// TIA Portal project "Data Logging Test 2_V17" (V17)

(* hardware
DEVICE "S7-1200 station_1"  S7-1200 Station
   slot 0: "Rack_0"  S7-1200 Rack  Rack  V1.0
   slot 1: "PLC_Wind Project-Datalogging"  CPU 1214C DC/DC/DC  6ES7 214-1AG40-0XB0  V4.2
   slot 2: "AI 4x13BIT/AQ 2x14BIT_1"  6ES7 234-4HE32-0XB0  V2.1
*)

// ===== PLC "PLC_Wind Project-Datalogging"  CPU 1214C DC/DC/DC =====

VAR_GLOBAL   // PLC tag table "Default tag table"
   "Enable_Write" AT %M10.0 : Bool;
   "Tag_2" AT %MD1 : DWord;
   "Potentiometer_Output" AT %MD6 : UDInt;
   "System_Byte" AT %MB1 : Byte;
   "FirstScan" AT %M1.0 : Bool;
   "DiagStatusUpdate" AT %M1.1 : Bool;
   "AlwaysTRUE" AT %M1.2 : Bool;
   "AlwaysFALSE" AT %M1.3 : Bool;
   "Clock_Byte" AT %MB0 : Byte;
   "Clock_10Hz" AT %M0.0 : Bool;
   "Clock_5Hz" AT %M0.1 : Bool;
   "Clock_2.5Hz" AT %M0.2 : Bool;
   "Clock_2Hz" AT %M0.3 : Bool;
   "Clock_1.25Hz" AT %M0.4 : Bool;
   "Clock_1Hz" AT %M0.5 : Bool;
   "Clock_0.625Hz" AT %M0.6 : Bool;
   "Clock_0.5Hz" AT %M0.7 : Bool;
   "Wind_Controller_Output" AT %MD12 : UDInt;
   "Enable_Wind_Write" AT %M10.1 : Bool;
   "Tag_1" AT %M10.4 : Bool;
END_VAR

VAR_GLOBAL   // PLC tag table "Tag table_1"
   "Start" AT %I1.0 : Bool;
   "Motor" AT %Q0.1 : Bool;
   "Green_LED" AT %Q0.3 : Bool;
   "Red_LED" AT %Q0.0 : Bool;
   "Potentiometer" AT %IW64 : Int;
   "Wind_Turbine_Controller" AT %IW96 : Int;
   "Start-Wind" AT %I0.2 : Bool;
END_VAR

DATA_BLOCK "wind"   // DB5
{ S7_Optimized_Access := 'TRUE' }
VERSION : 0.1
   VAR
      records : UDInt := 50;
      "name" : String := 'OutputVoltage';
      id : DWord := 2;
      headers : String := 'Vout';
      data : Struct
         "Output Voltage" : UDInt;
      END_STRUCT;
      done : Bool;
      busy : Bool;
      error : Bool;
      status : Word;
   END_VAR
BEGIN
END_DATA_BLOCK

FUNCTION "WindController_Config" : Void   // FC2, LAD
TITLE = CONFIGURING ANALOG SENSOR - WIND CONTROLLER
{ S7_Optimized_Access := 'TRUE' }
VERSION : 0.1
// USE OF NORM_X AND SCALE_X BLOCKS
   VAR_INPUT
      Input_Wind_Norm : Int;
   END_VAR
   VAR_OUTPUT
      Output_Wind_Scaled : UDInt;
   END_VAR
   VAR_TEMP
      Output_Wind_Norm : Real;
   END_VAR
BEGIN

REGION Network 1: NORM_X
   // CONVERSION OF PLC BIT VALUES FROM INT TO REAL VALUES THAT CAN BE SCALED/ LINEARIZED
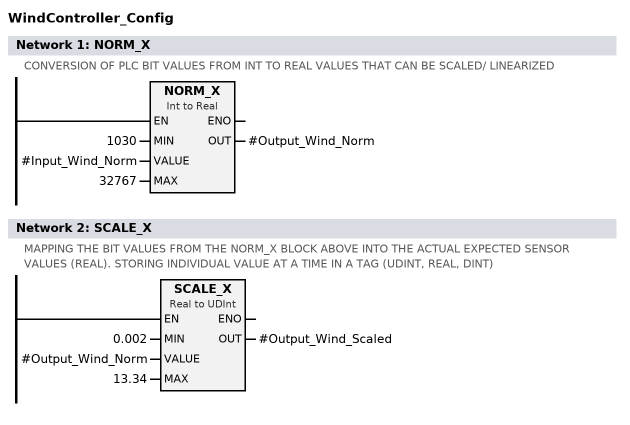
   RUNG wire#powerrail
      { S7_Templates := "[SrcType := Int, DestType := Real]" } Normalize(min := 1030, value := #Input_Wind_Norm, max := 32767, out => #Output_Wind_Norm)
   END_RUNG
   // the same network as SCL:
   #Output_Wind_Norm := NORM_X(MIN := 1030, VALUE := #Input_Wind_Norm, MAX := 32767);
END_REGION

REGION Network 2: SCALE_X
   // MAPPING THE BIT VALUES FROM THE NORM_X BLOCK ABOVE INTO THE ACTUAL EXPECTED SENSOR VALUES (REAL). STORING INDIVIDUAL VALUE AT A TIME IN A TAG (UDINT, REAL, DINT)
   RUNG wire#powerrail
      { S7_Templates := "[SrcType := Real, DestType := UDInt]" } Scale(min := 0.002, value := #Output_Wind_Norm, max := 13.34, out => #Output_Wind_Scaled)
   END_RUNG
   // the same network as SCL:
   #Output_Wind_Scaled := SCALE_X(MIN := 0.002, VALUE := #Output_Wind_Norm, MAX := 13.34);
END_REGION
END_FUNCTION

ORGANIZATION_BLOCK "Main"   // OB1, LAD, ProgramCycle
TITLE = "Main Program Sweep (Cycle)"
{ S7_Optimized_Access := 'TRUE' }
VERSION : 0.1
// RUN THE WIND CONTROLLER CONFIGURATION. PERFORM DATALOGGING WHICH ENTAILS DATALOG CREATE AND DATALOG WRITE BLOCK FROM THE EXTENDED INSTRUCTIONS(RECIPE & DATA LOGGING)
   VAR_INPUT
      Initial_Call : Bool;   // Initial call of this OB
      Remanence : Bool;   // =True, if remanent data are available
   END_VAR
BEGIN

REGION Network 1: PULL THE WIND CONROLLER CONFIG FUNCTION IN
   // FULL EXECUTION OF NORM_X AND SCALE_X FOR OUR SENSOR
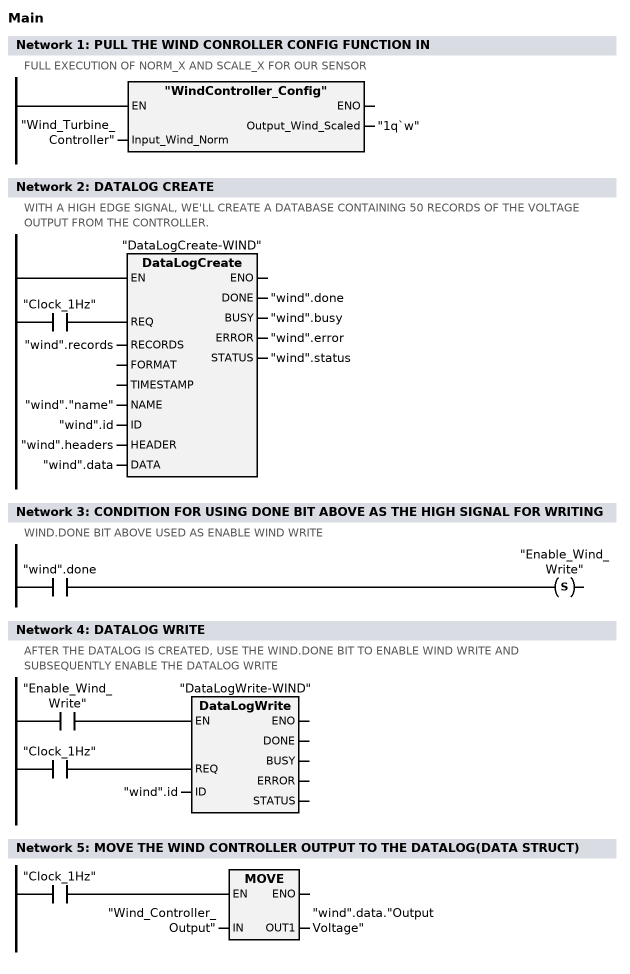
   RUNG wire#powerrail
      "WindController_Config"(Input_Wind_Norm := "Wind_Turbine_Controller", Output_Wind_Scaled => "1q`w")
   END_RUNG
   // the same network as SCL:
   "WindController_Config"(Input_Wind_Norm := "Wind_Turbine_Controller", Output_Wind_Scaled => "1q`w");
END_REGION

REGION Network 2: DATALOG CREATE
   // WITH A HIGH EDGE SIGNAL, WE'LL CREATE A DATABASE CONTAINING 50 RECORDS OF THE VOLTAGE OUTPUT FROM THE CONTROLLER.
   "DataLogCreate-WIND"(REQ := "Clock_1Hz",   // DataLogCreate
                        RECORDS := "wind".records,
                        "NAME" := "wind"."name",
                        ID := "wind".id,
                        HEADER := "wind".headers,
                        DATA := "wind".data,
                        DONE => "wind".done,
                        BUSY => "wind".busy,
                        ERROR => "wind".error,
                        STATUS => "wind".status);
END_REGION

REGION Network 3: CONDITION FOR USING DONE BIT ABOVE AS THE HIGH SIGNAL FOR WRITING
   // WIND.DONE BIT ABOVE USED AS ENABLE WIND WRITE
   RUNG wire#powerrail
      Contact( "wind".done )
      S_Coil( "Enable_Wind_Write" )
   END_RUNG
   // the same network as SCL:
   IF "wind".done THEN "Enable_Wind_Write" := TRUE; END_IF;
END_REGION

REGION Network 4: DATALOG WRITE
   // AFTER THE DATALOG IS CREATED, USE THE WIND.DONE BIT TO ENABLE WIND WRITE AND SUBSEQUENTLY ENABLE THE DATALOG WRITE
   IF "Enable_Wind_Write" THEN
       "DataLogWrite-WIND"(REQ := "Clock_1Hz", ID := "wind".id);   // DataLogWrite
   END_IF;
END_REGION

REGION Network 5: MOVE THE WIND CONTROLLER OUTPUT TO THE DATALOG(DATA STRUCT)
   RUNG wire#powerrail
      Contact( "Clock_1Hz" )
      Move(in := "Wind_Controller_Output", out1 => "wind".data."Output Voltage")
   END_RUNG
   // the same network as SCL:
   IF "Clock_1Hz" THEN "wind".data."Output Voltage" := "Wind_Controller_Output"; END_IF;
END_REGION
END_ORGANIZATION_BLOCK